// TIA Portal V20 export
TYPE "type_emRelations_em1_SoftCam"
// stored: Access Published, Namespace Unit1
   STRUCT
      unwinderBtmAxisB : Struct
         Pos00 { S7_SetPoint := 'True'} : "LER_typeSoftCamPosition";
         Pos01 { S7_SetPoint := 'True'} : "LER_typeSoftCamPosition";
         Pos02 { S7_SetPoint := 'True'} : "LER_typeSoftCamPosition";
         Pos03 { S7_SetPoint := 'True'} : "LER_typeSoftCamPosition";
         Pos04 { S7_SetPoint := 'True'} : "LER_typeSoftCamPosition";
         Pos05 { S7_SetPoint := 'True'} : "LER_typeSoftCamPosition";
         Pos06 { S7_SetPoint := 'True'} : "LER_typeSoftCamPosition";
         Pos07 { S7_SetPoint := 'True'} : "LER_typeSoftCamPosition";
         Pos08 { S7_SetPoint := 'True'} : "LER_typeSoftCamPosition";
         Pos09 { S7_SetPoint := 'True'} : "LER_typeSoftCamPosition";
         Pos10 { S7_SetPoint := 'True'} : "LER_typeSoftCamPosition";
         Pos11 { S7_SetPoint := 'True'} : "LER_typeSoftCamPosition";
         Pos12 { S7_SetPoint := 'True'} : "LER_typeSoftCamPosition";
         Pos13 { S7_SetPoint := 'True'} : "LER_typeSoftCamPosition";
         Pos14 { S7_SetPoint := 'True'} : "LER_typeSoftCamPosition";
         Pos15 { S7_SetPoint := 'True'} : "LER_typeSoftCamPosition";
      END_STRUCT;
   END_STRUCT;
END_TYPE
